(* IEC 61131-3 sources: lasal-git-demo/CPU/LasalDemoProject/Class/OPC_UA_Interface, 1 file *)

(* ---- OPC_UA_Interface.st ---- *)
(*!
<Class
	Name               = "OPC_UA_Interface"
	Revision           = "1.1"
	RealtimeTask       = "false"
	CyclicTask         = "false"
	BackgroundTask     = "false"
	Sigmatek           = "true"
	OSInterface        = "false"
	HighPriority       = "false"
	Automatic          = "false"
	UpdateMode         = "Prescan"
	SharedCommandTable = "true"
	Objectsize         = "(396,120)">
	<Channels>
		<Server Name="ClassSvr" Visualized="false" Initialize="false" WriteProtected="true" Retentive="false"/>
		<Client Name="OPC_UA" Required="true" Internal="false"/>
	</Channels>
	<RevDoku>
		<Owner Company="Sigmatek"/>
		<Dokumentation Revision="1.1" Date="2019-07-30" Author="FurLuk" Company="Sigmatek" Description="Added Callback Methods with ApplicationUri when a Client is creating and closing a session"/>
		<Dokumentation Revision="1.0" Date="2019-07-30" Author="HubChr" Company="Sigmatek" Description="Creation"/>
	</RevDoku>
</Class>
*)
OPC_UA_Interface : CLASS
  //Servers:
	ClassSvr 	: SvrChCmd_DINT;
  //Clients:
	OPC_UA 	: CltChCmd_OPC_UA;
  //Variables:
		usInitCnt 	: DINT;
  //Functions:

	FUNCTION VIRTUAL GLOBAL Init;
				//! <Function Comment="Callback to the application. Is called each time an application certificate is activated, &#13;&#10;e.g. after booting or after creating a certificate via CreateApplCertificate()." Name="CB_CertificateLoaded"/>
	FUNCTION VIRTUAL GLOBAL CB_CertificateLoaded
		VAR_INPUT
			IF_Number 	: UDINT;
			ValidTo 	: DINT;
		END_VAR
		VAR_OUTPUT
			retcode 	: DINT;
		END_VAR;
				//! <Function Comment="Callback to the application. Called when a new certificate is to be validated.&#13;&#10;The response can be made using the CertificateValidationFeedback () method." Name="CB_ValidateCertificate"/>
	FUNCTION VIRTUAL GLOBAL CB_ValidateCertificate
		VAR_INPUT
			certificateInfo 	: OPC_UA::ptrOpcUa_PkiCertificateInfo;
			identity 	: OPC_UA::ptrOpcUa_PkiIdentity;
			fileName 	: ^CHAR;
			certificateData 	: ^BYTE;
			certificateLength 	: DINT;
		END_VAR
		VAR_OUTPUT
			retcode 	: DINT;
		END_VAR;
				//! <Function Comment="Callback to the application.&#13;&#10;Is called each time a Client is creating a session." Name="CB_CreateSession"/>
	FUNCTION VIRTUAL GLOBAL CB_CreateSession
		VAR_INPUT
			pApplicationUri 	: ^void;			//! <Variable Comment="pointer to the ApplicationUri of the client information" Name="CB_CreateSession.pApplicationUri"/>
		END_VAR;
				//! <Function Comment="Callback to the application.&#13;&#10;Is called each time a Client is closing a session." Name="CB_CloseSession"/>
	FUNCTION VIRTUAL GLOBAL CB_CloseSession
		VAR_INPUT
			pApplicationUri 	: ^void;			//! <Variable Comment="pointer to the ApplicationUri of the client information" Name="CB_CloseSession.pApplicationUri"/>
		END_VAR;
  //Tables:
	FUNCTION @STD
		VAR_OUTPUT
			ret_code	: CONFSTATES;
		END_VAR;
	FUNCTION GLOBAL TAB @CT_;
END_CLASS;

#pragma usingLtd OPC_UA

FUNCTION VIRTUAL GLOBAL OPC_UA_Interface::Init

  if usInitCnt = 1 then
    OPC_UA.RegisterInterfaceClass(this);
  end_if;

  usInitCnt += 1;

END_FUNCTION

#pragma warning(disable:73);
FUNCTION VIRTUAL GLOBAL OPC_UA_Interface::CB_CertificateLoaded
	VAR_INPUT
		IF_Number 	: UDINT;
		ValidTo 	: DINT;
	END_VAR
	VAR_OUTPUT
		retcode 	: DINT;
	END_VAR

  retcode := 0;

END_FUNCTION
#pragma warning(default:73);

#pragma warning(disable:73);
FUNCTION VIRTUAL GLOBAL OPC_UA_Interface::CB_ValidateCertificate
	VAR_INPUT
		certificateInfo 	: OPC_UA::ptrOpcUa_PkiCertificateInfo;
		identity 	: OPC_UA::ptrOpcUa_PkiIdentity;
		fileName 	: ^CHAR;
		certificateData 	: ^BYTE;
		certificateLength 	: DINT;
	END_VAR
	VAR_OUTPUT
		retcode 	: DINT;
	END_VAR

  // activate for auto-trusting
  // retcode := CertificateValidationFeedback(fileName, certificateData, certificateLength, Trust);

  retcode := 0;

END_FUNCTION
#pragma warning(default:73);

#pragma warning(disable:73);
FUNCTION VIRTUAL GLOBAL OPC_UA_Interface::CB_CreateSession
	VAR_INPUT
		pApplicationUri 	: ^void;
	END_VAR

END_FUNCTION
#pragma warning(default:73);

#pragma warning(disable:73);
FUNCTION VIRTUAL GLOBAL OPC_UA_Interface::CB_CloseSession
	VAR_INPUT
		pApplicationUri 	: ^void;
	END_VAR

END_FUNCTION
#pragma warning(default:73);
